// TIA Portal V19 export
FUNCTION "Output Force to auto" : Void   // FC31, STL
{ S7_Optimized_Access := 'TRUE' }
AUTHOR : JOM
FAMILY : APP
NAME : FORCE
// FORCE ALL OUTPUTS INTO AUTOMATIC MODE
// stored: AutoNumber false
BEGIN

NETWORK
TITLE = 
// OUTPUTS CARD 1
      SET;
      S     "ItemCommand".Y0101.Auto;
      S     "ItemCommand".Y0103.Auto;
      S     "ItemCommand".Y0104.Auto;
      S     "ItemCommand".Y0109.Auto;
      S     "ItemCommand".Y0111.Auto;
      S     "ItemCommand".Y0112.Auto;
      S     "ItemCommand".Y0113.Auto;
      S     "ItemCommand".Y0114.Auto;
      S     "ItemCommand".Y0115.Auto;
      S     "ItemCommand".M0139.Auto;
      S     "ItemCommand".Y0116.Auto;
      S     "ItemCommand".Y0108.Auto;
      S     "ItemCommand".Y0117.Auto;
      S     "ItemCommand".Y0118.Auto;
      S     "ItemCommand".Y0237.Auto;
      S     "ItemCommand".Y0238.Auto;

NETWORK
TITLE = 
// OUTPUTS CARD 2
      S     "ItemCommand".Y0119.Auto;
      S     "ItemCommand".Y0124.Auto;
      S     "ItemCommand".Y0135_NOT_USED.Auto;
      S     "ItemCommand".Y0136_NOT_USED.Auto;
      S     "ItemCommand".Y0137_NOT_USED.Auto;
      S     "ItemCommand".Y0143.Auto;
      S     "ItemCommand".Y0144_NOT_USED.Auto;
      S     "ItemCommand".Y0147.Auto;
      S     "ItemCommand".Y0148.Auto;
      S     "ItemCommand".Y0158.Auto;
      S     "ItemCommand".Y0545.Auto;
      S     "ItemCommand".PACK1.Auto;
      S     "ItemCommand".PACK2.Auto;
      S     "ItemCommand".PACK3.Auto;
      S     "ItemCommand".PACK4.Auto;
      S     "ItemCommand".AlarmLamp.Auto;

NETWORK
TITLE = 
// OUTPUTS CARD 3
      S     "ItemCommand".AHV_CLOSED.Auto;
      S     "ItemCommand".AHV_HIGH_LEVEL.Auto;
      S     "ItemCommand".AHV_READY.Auto;
      S     "ItemCommand".AHV_SHUT_DOWN.Auto;
      S     "ItemCommand".AHV_STERILE.Auto;
      S     "ItemCommand".PROD_AVAILABLE.Auto;
      S     "ItemCommand".RINSE_READY.Auto;
      S     "ItemCommand".CAUSTIC_READY.Auto;
      S     "ItemCommand".ACID_READY.Auto;
      S     "ItemCommand".CIP_FILLER_ENABLE.Auto;
      S     "ItemCommand".WATER_PUMP.Auto;
      S     "ItemCommand".Y0901.Auto;
      S     "ItemCommand".Y0902.Auto;
      S     "ItemCommand".Y0903.Auto;
      S     "ItemCommand".TANK_READY.Auto;
      S     "ItemCommand".TANK_OPEN.Auto;

NETWORK
TITLE = 
      S     "ItemCommand".Y0904.Auto;
      S     "ItemCommand".Y0905.Auto;
      S     "ItemCommand".Y0906.Auto;
      S     "ItemCommand".Y0907.Auto;
      S     "ItemCommand".Y0908.Auto;
      S     "ItemCommand".Y0909.Auto;
      S     "ItemCommand".Y0910.Auto;
      S     "ItemCommand".Y0911.Auto;
      S     "ItemCommand".Y0912.Auto;
      S     "ItemCommand".Q41_1.Auto;
      S     "ItemCommand".CIP_Route.Auto;
      S     "ItemCommand".SIP_Steam.Auto;
      S     "ItemCommand".Product_Available.Auto;
      S     "ItemCommand".Barrier_Sterile.Auto;
      S     "ItemCommand".Product_Route.Auto;
      S     "ItemCommand".X0913.Auto;
END_FUNCTION
